// TIA Portal V20 export
DATA_BLOCK "AlarmTrigger"   // DB7
{ S7_Optimized_Access := 'TRUE' }
// stored: MemoryReserve 100
   VAR
      TriggerTag : Bool;
   END_VAR
BEGIN
END_DATA_BLOCK
